# EPICS autosave request: mcaApp/Db/Amptek_settings.req
$(P)$(R)InputPolarity
$(P)$(R)Clock
$(P)$(R)Gain
$(P)$(R)Gate
$(P)$(R)PeakingTime
$(P)$(R)FastPeakingTime
$(P)$(R)FlatTopTime
$(P)$(R)SlowThreshold
$(P)$(R)FastThreshold
$(P)$(R)PUREnable
$(P)$(R)MCASource
$(P)$(R)ConfigFileName
$(P)$(R)ReadStatus.SCAN
$(P)$(R)SetDetTemp
$(P)$(R)SetHighVoltage
